// Mitsubishi GX Works2 project: somatoria   PLC: Q03UDV

PROGRAM MAIN
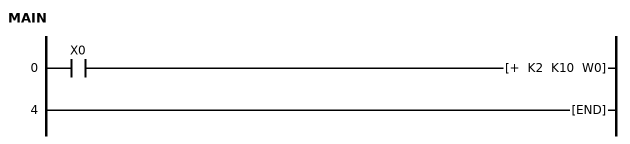
0     LD      X0
      +       K2 K10 W0
4     END
END_PROGRAM
